KUKA KRL data list: check_game_over.dat

&ACCESS RV1
DEFDAT  check_game_over PUBLIC

ENDDAT
